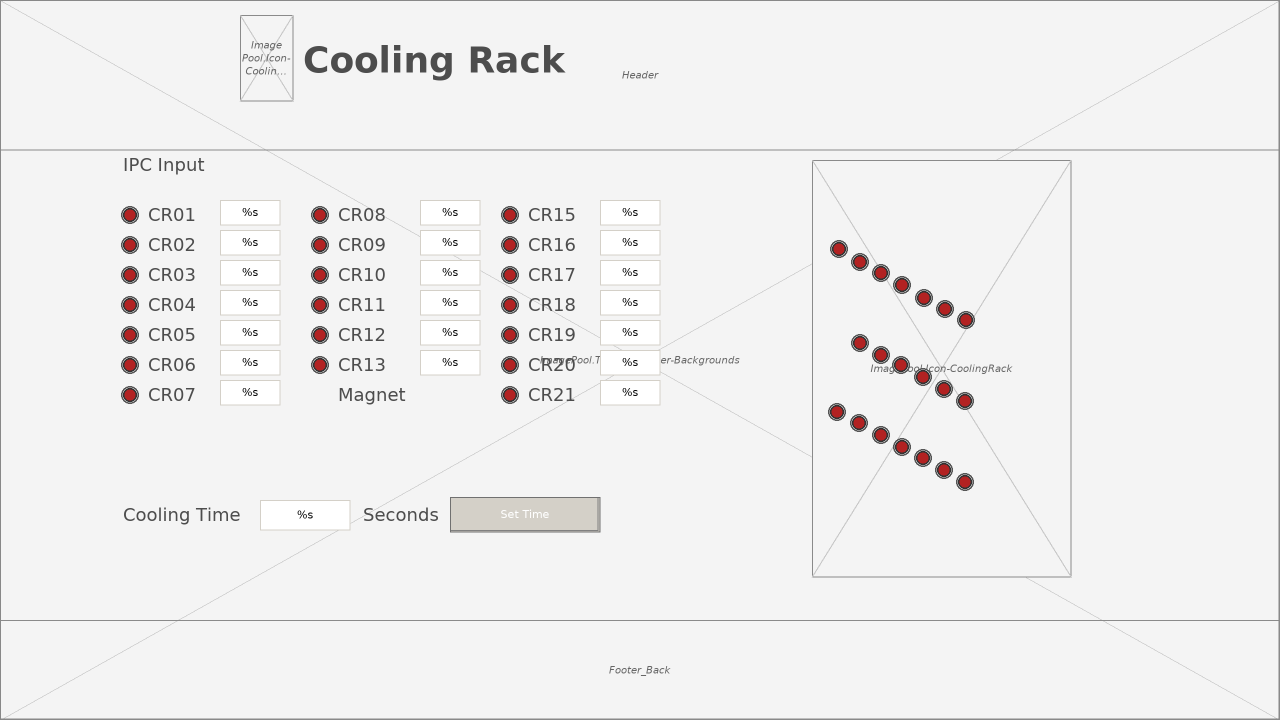
VISUALIZATION PAGE_CoolRack  // 1280x720
    Image (0,0 1280x720), image: ImagePool.The-New-Silver-Backgrounds
    Frame (0,620 1280x100)
        shows Footer_Back()
    Frame (0,0 1280x150)
        shows Header()
    Label (300,40 300x40), "Cooling Rack"
    Label (145,200 60x30), "CR01"
    Label (145,230 60x30), "CR02"
    Label (145,260 60x30), "CR03"
    Label (145,290 60x30), "CR04"
    Label (145,320 60x30), "CR05"
    Lamp1 (120,325 20x20), variable: COOL_RACK.CR[5], style: Lamp-Lamp1-Red
    Label (145,350 60x30), "CR06"
    Lamp1 (120,355 20x20), variable: COOL_RACK.CR[6], style: Lamp-Lamp1-Red
    Label (145,380 60x30), "CR07"
    Lamp1 (120,385 20x20), variable: COOL_RACK.CR[7], style: Lamp-Lamp1-Red
    Label (120,150 150x30), "IPC Input"
    Image (240,15 53x86), image: ImagePool.Icon-CoolingRack
    Image (812,160 259x417), image: ImagePool.Icon-CoolingRack
    Lamp1 (956,310 20x20), variable: COOL_RACK.CR[1], style: Lamp-Lamp1-Red
    Lamp1 (935,299 20x20), variable: COOL_RACK.CR[2], style: Lamp-Lamp1-Red
    Lamp1 (914,288 20x20), variable: COOL_RACK.CR[3], style: Lamp-Lamp1-Red
    Lamp1 (892,275 20x20), variable: COOL_RACK.CR[4], style: Lamp-Lamp1-Red
    Lamp1 (871,263 20x20), variable: COOL_RACK.CR[5], style: Lamp-Lamp1-Red
    Lamp1 (850,252 20x20), variable: COOL_RACK.CR[6], style: Lamp-Lamp1-Red
    Lamp1 (829,239 20x20), variable: COOL_RACK.CR[7], style: Lamp-Lamp1-Red
    Lamp1 (934,379 20x20), variable: COOL_RACK.CR[9], style: Lamp-Lamp1-Red
    Lamp1 (955,391 20x20), variable: COOL_RACK.CR[8], style: Lamp-Lamp1-Red
    Lamp1 (913,367 20x20), variable: COOL_RACK.CR[10], style: Lamp-Lamp1-Red
    Lamp1 (891,355 20x20), variable: COOL_RACK.CR[11], style: Lamp-Lamp1-Red
    Lamp1 (871,345 20x20), variable: COOL_RACK.CR[12], style: Lamp-Lamp1-Red
    Lamp1 (850,333 20x20), variable: COOL_RACK.CR[13], style: Lamp-Lamp1-Red
    Lamp1 (955,472 20x20), variable: COOL_RACK.CR[15], style: Lamp-Lamp1-Red
    Lamp1 (934,460 20x20), variable: COOL_RACK.CR[16], style: Lamp-Lamp1-Red
    Lamp1 (913,448 20x20), variable: COOL_RACK.CR[17], style: Lamp-Lamp1-Red
    Lamp1 (892,437 20x20), variable: COOL_RACK.CR[18], style: Lamp-Lamp1-Red
    Lamp1 (871,425 20x20), variable: COOL_RACK.CR[19], style: Lamp-Lamp1-Red
    Lamp1 (849,413 20x20), variable: COOL_RACK.CR[20], style: Lamp-Lamp1-Red
    Lamp1 (827,402 20x20), variable: COOL_RACK.CR[21], style: Lamp-Lamp1-Red
    Label (120,500 150x30), "Cooling Time"
    Textfield (260,500 90x30), "%s", text variable: GVL.iCooling_Time
        OnMouseClick: write the text variable via VisuDialogs.Numpad, min 1, max 1000, title 'Cooling Time (min)'
    Textfield (220,200 60x25), "%s", text variable: GVL.CRTimer[1]
    Textfield (220,230 60x25), "%s", text variable: GVL.CRTimer[2]
    Textfield (220,260 60x25), "%s", text variable: GVL.CRTimer[3]
    Textfield (220,290 60x25), "%s", text variable: GVL.CRTimer[4]
    Textfield (220,320 60x25), "%s", text variable: GVL.CRTimer[5]
    Textfield (220,350 60x25), "%s", text variable: GVL.CRTimer[6]
    Textfield (220,380 60x25), "%s", text variable: GVL.CRTimer[7]
    Label (335,200 60x30), "CR08"
    Lamp1 (310,205 20x20), variable: COOL_RACK.CR[8], style: Lamp-Lamp1-Red
    Label (335,230 60x30), "CR09"
    Lamp1 (310,235 20x20), variable: COOL_RACK.CR[9], style: Lamp-Lamp1-Red
    Label (335,260 60x30), "CR10"
    Lamp1 (310,265 20x20), variable: COOL_RACK.CR[10], style: Lamp-Lamp1-Red
    Label (335,290 60x30), "CR11"
    Lamp1 (310,295 20x20), variable: COOL_RACK.CR[11], style: Lamp-Lamp1-Red
    Label (335,320 60x30), "CR12"
    Lamp1 (310,325 20x20), variable: COOL_RACK.CR[12], style: Lamp-Lamp1-Red
    Label (335,350 60x30), "CR13"
    Lamp1 (310,355 20x20), variable: COOL_RACK.CR[13], style: Lamp-Lamp1-Red
    Label (335,380 91x30), "Magnet"
    Textfield (420,230 60x25), "%s", text variable: GVL.CRTimer[9]
    Textfield (420,200 60x25), "%s", text variable: GVL.CRTimer[8]
    Textfield (420,260 60x25), "%s", text variable: GVL.CRTimer[10]
    Textfield (420,290 60x25), "%s", text variable: GVL.CRTimer[11]
    Textfield (420,320 60x25), "%s", text variable: GVL.CRTimer[12]
    Textfield (420,350 60x25), "%s", text variable: GVL.CRTimer[13]
    Label (525,200 60x30), "CR15"
    Lamp1 (500,205 20x20), variable: COOL_RACK.CR[15], style: Lamp-Lamp1-Red
    Label (525,230 60x30), "CR16"
    Lamp1 (500,235 20x20), variable: COOL_RACK.CR[16], style: Lamp-Lamp1-Red
    Label (525,260 60x30), "CR17"
    Lamp1 (500,265 20x20), variable: COOL_RACK.CR[17], style: Lamp-Lamp1-Red
    Label (525,290 60x30), "CR18"
    Lamp1 (500,295 20x20), variable: COOL_RACK.CR[18], style: Lamp-Lamp1-Red
    Label (525,320 60x30), "CR19"
    Lamp1 (500,325 20x20), variable: COOL_RACK.CR[19], style: Lamp-Lamp1-Red
    Label (525,350 60x30), "CR20"
    Lamp1 (500,355 20x20), variable: COOL_RACK.CR[20], style: Lamp-Lamp1-Red
    Label (525,380 60x30), "CR21"
    Lamp1 (500,385 20x20), variable: COOL_RACK.CR[21], style: Lamp-Lamp1-Red
    Textfield (600,230 60x25), "%s", text variable: GVL.CRTimer[16]
    Textfield (600,200 60x25), "%s", text variable: GVL.CRTimer[15]
    Textfield (600,260 60x25), "%s", text variable: GVL.CRTimer[17]
    Textfield (600,290 60x25), "%s", text variable: GVL.CRTimer[18]
    Textfield (600,320 60x25), "%s", text variable: GVL.CRTimer[19]
    Textfield (600,350 60x25), "%s", text variable: GVL.CRTimer[20]
    Textfield (600,380 60x25), "%s", text variable: GVL.CRTimer[21]
    Button (450,497 150x35), "Set Time"
        tap COOL_RACK.set_time
    Label (360,500 80x30), "Seconds"
    Lamp1 (120,205 20x20), variable: COOL_RACK.CR[1], style: Lamp-Lamp1-Red
    Lamp1 (120,235 20x20), variable: COOL_RACK.CR[2], style: Lamp-Lamp1-Red
    Lamp1 (120,265 20x20), variable: COOL_RACK.CR[3], style: Lamp-Lamp1-Red
    Lamp1 (120,295 20x20), variable: COOL_RACK.CR[4], style: Lamp-Lamp1-Red
END_VISUALIZATION

(* stored: Version 1.1.0.1, ProductVersion 3.1.4024.12
   Visu PAGE_CoolRack: Id {c78cd257-5751-48bb-a7ea-e5c18da7b8d4} *)
